FUNCTION F_tanh : LREAL
VAR_INPUT
	x: LREAL;
END_VAR

F_tanh := (EXP(x) - EXP(-x))/(EXP(x) + EXP(-x));

END_FUNCTION

(* stored: Version 1.1.0.1, ProductVersion 3.1.4024.12
   POU F_tanh: Id {df10c944-7ba5-44b6-bd6b-400e6c78d620}, SpecialFunc None *)
